FUNCTION_BLOCK INT_TRIGGER (* Composite Function Block Type *)
  (* Standard: 61499-2 *)
  (* Version 1.0, 2019-02-10, iotdeveloperpk *)
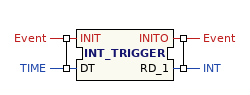
  EVENT_INPUT
    INIT WITH DT; (* Initialization Request *)
  END_EVENT
  EVENT_OUTPUT
    INITO WITH RD_1; (* Initialization Confirm *)
  END_EVENT
  VAR_INPUT
    DT : TIME;
  END_VAR
  VAR_OUTPUT
    RD_1 : INT;
  END_VAR
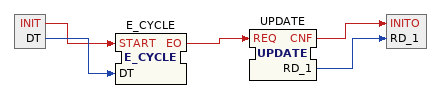
  FBS
    UPDATE : UPDATE;
    E_CYCLE : E_CYCLE;
  END_FBS
  EVENT_CONNECTIONS
    E_CYCLE.EO TO UPDATE.REQ;
    INIT TO E_CYCLE.START;
    UPDATE.CNF TO INITO;
  END_CONNECTIONS
  DATA_CONNECTIONS
    UPDATE.RD_1 TO RD_1;
    DT TO E_CYCLE.DT;
  END_CONNECTIONS
END_FUNCTION_BLOCK
